// TIA Portal V17 export
// export: Created 2022-07-16T16:56:13.3756579Z, ExportSetting WithDefaults, DisplayName Totally Integrated Automation Portal, DisplayVersion V17, DisplayName TIA Portal Openness, DisplayVersion V17, DisplayName TIA Portal Version Control Interface, DisplayVersion V17, DisplayName TIA Portal Test Suite Advanced, DisplayVersion V17, DisplayName STEP 7 Professional, DisplayVersion V17, DisplayName STEP 7 Safety, DisplayVersion V17, DisplayName WinCC Professional, DisplayVersion V17
TYPE "Client interface_1.dbData.postTestResult.preTestCheckSequence.pressures"
// stored: IsFailsafeCompliant false
   STRUCT
      validation { ExternalWritable := 'False'; S7_SetPoint := 'True'} : "Client interface_1.dbData.postTestResult.preTestCheckSequence.pressures.validation";
      airHoldTest { ExternalWritable := 'False'; S7_SetPoint := 'True'} : "Client interface_1.dbData.postTestResult.preTestCheckSequence.pressures.airHoldTest";
      drainTest { ExternalWritable := 'False'; S7_SetPoint := 'True'} : "Client interface_1.dbData.postTestResult.preTestCheckSequence.pressures.drainTest";
   END_STRUCT;
END_TYPE
